FUNCTION_BLOCK ReactorInStatus (* Basic Function Block Type *)
  (* Standard: 61499-2 *)
  (* Version 0.0, 7/31/2026, Schneider Electric, Template *)
  PACKAGE SE.Nereda;
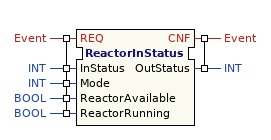
  EVENT_INPUT
    REQ WITH InStatus, ReactorAvailable, ReactorRunning, Mode; (* Normal Execution Request *)
  END_EVENT
  EVENT_OUTPUT
    CNF WITH OutStatus; (* Execution Confirmation *)
  END_EVENT
  VAR_INPUT
    InStatus : INT;
    Mode : INT;
    ReactorAvailable : BOOL;
    ReactorRunning : BOOL;
  END_VAR
  VAR_OUTPUT
    OutStatus : INT;
  END_VAR
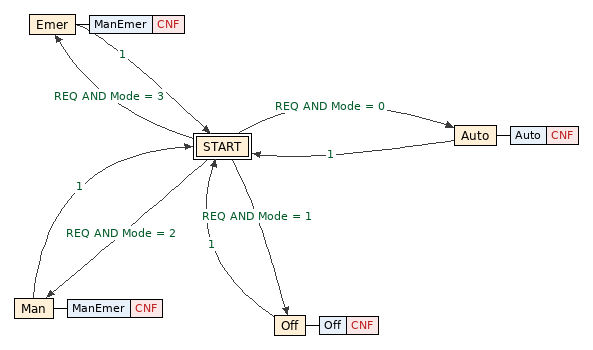
  EC_STATES
    START; (* Initial State *)
    Auto : Auto -> CNF; (* Initialization *)
    Off : Off -> CNF; (* Normal execution *)
    Man : ManEmer -> CNF;
    Emer : ManEmer -> CNF;
  END_STATES
  EC_TRANSITIONS
    START TO Auto := REQ AND Mode = 0;
    Auto TO START := 1;
    START TO Off := REQ AND Mode = 1;
    Off TO START := 1;
    START TO Man := REQ AND Mode = 2;
    Man TO START := 1;
    START TO Emer := REQ AND Mode = 3;
    Emer TO START := 1;
  END_TRANSITIONS
  ALGORITHM Emer IN ST: (* Normally executed algorithm *)
;
  END_ALGORITHM
  ALGORITHM Auto IN ST:
;
OutStatus := InStatus;
  END_ALGORITHM
  ALGORITHM Off IN ST:
;
OutStatus := 10;
  END_ALGORITHM
  ALGORITHM ManEmer IN ST:
;
IF NOT ReactorRunning AND NOT ReactorAvailable THEN
	OutStatus := 6;
ELSIF NOT ReactorRunning AND ReactorAvailable THEN
	OutStatus := 0;
ELSIF ReactorRunning AND NOT ReactorAvailable THEN
	OutStatus := 6;
ELSIF ReactorRunning AND ReactorAvailable THEN
	OutStatus := 2;
END_IF;
  END_ALGORITHM
END_FUNCTION_BLOCK
